Staubli VAL3: trajectory.dtx

public string sItems
string sPath = "Disk://saveTraj/"
public bool bMoveType[3]
public bool bStepping
